(* IEC 61131-3 sources: Mizera_Tube/Plc (part 8) *)

END_VAR

VAR_OUTPUT
yax_READY:    BOOL;       * FB pronto per START
yax_RUNNING:  BOOL;       * Esecuzione FB in corso
yax_ENDOK:    BOOL;       * Comando terminato correttamente
yax_ENDERR:   BOOL;       * Comando terminato non correttamente
yax_ERRCODE:  DWORD;      * codice errore ( maschera bit )
END_VAR

VAR
AXFB: AX_COMMAND;
END_VAR

* Chiamata FB standard gestione comandi slave

LD   xax_ENABLE                    ** abilita FB
ST   AXFB.xax_ENABLE

LD   xax_START                     ** start richiesta azione
ST   AXFB.xax_START

LD   xax_CLEAR                     ** conferma fine comando
ST   AXFB.xax_CLEAR

CAL  AXFB

* Comando uscite da FB standard

LD   AXFB.yax_READY
ST   yax_READY                     ** FB pronto per START

LD   AXFB.yax_RUNNING
ST   yax_RUNNING                   ** Esecuzione FB in corso

LD   AXFB.yax_ENDOK
ST   yax_ENDOK                     ** Comando terminato correttamente

LD   AXFB.yax_ENDERR
ST   yax_ENDERR                    ** Comando terminato non correttamente

LD   AXFB.yax_ERRCODE
ST   yax_ERRCODE                   ** codice errore ( maschera bit )

*** TRASFERIMENTO DEI REGISTRI FB ALLO SLAVE ***

LD   AXFB.yax_RUNSLV
JMPCN END_DATA

LD   29
ST   FB_CODE                       ** fb0 Codice Operativo comando

LD   xax_NODE                      ** Numero nodo richiesto (2-60) o maschera
ST   %fb1

LD   xax_MODE                      ** Tipo di comando
ST   %fb2

END_DATA:

END_FUNCTION_BLOCK

* ----------------------------------------------------*
* Blocco Funzionale abilita/disabilita operatore dinamico su un asse
* ----------------------------------------------------*

FUNCTION_BLOCK AX_COUP

VAR_INPUT
xax_ENABLE:   BOOL;       * abilita FB
xax_START:    BOOL;       * start richiesta azione
xax_CLEAR:    BOOL;       * conferma fine comando
xax_MODE:     DWORD;      * Funzione selezionata
xax_INSTANCE: DWORD;      * Numero istanza tabella dati
xax_MASTER0:  DWORD;      * Numero asse master 0
xax_MASTER1:  DWORD;      * Numero asse master 1
xax_MASTER2:  DWORD;      * Numero asse master 2
xax_MASTER3:  DWORD;      * Numero asse master 3
xax_MASTER4:  DWORD;      * Numero asse master 4
xax_MASTER5:  DWORD;      * Numero asse master 5

END_VAR

VAR_OUTPUT
yax_READY:    BOOL;       * FB pronto per START
yax_RUNNING:  BOOL;       * Esecuzione FB in corso
yax_ENDOK:    BOOL;       * Comando terminato correttamente
yax_ENDERR:   BOOL;       * Comando terminato non correttamente
yax_ERRCODE:  DWORD;      * codice errore ( maschera bit )
END_VAR

VAR
AXFB: AX_COMMAND;
END_VAR

* Chiamata FB standard gestione comandi slave

LD   xax_ENABLE                    ** abilita FB
ST   AXFB.xax_ENABLE

LD   xax_START                     ** start richiesta azione
ST   AXFB.xax_START

LD   xax_CLEAR                     ** conferma fine comando
ST   AXFB.xax_CLEAR

CAL  AXFB

* Comando uscite da FB standard

LD   AXFB.yax_READY
ST   yax_READY                     ** FB pronto per START

LD   AXFB.yax_RUNNING
ST   yax_RUNNING                   ** Esecuzione FB in corso

LD   AXFB.yax_ENDOK
ST   yax_ENDOK                     ** Comando terminato correttamente

LD   AXFB.yax_ENDERR
ST   yax_ENDERR                    ** Comando terminato non correttamente

LD   AXFB.yax_ERRCODE
ST   yax_ERRCODE                   ** codice errore ( maschera bit )

*** TRASFERIMENTO DEI REGISTRI FB ALLO SLAVE ***

LD   AXFB.yax_TRDATA
JMPCN END_DATA

LD   31
ST   FB_CODE                       ** fb0 Codice Operativo comando

LD   xax_MODE                      ** Funzione selezionata
ST   FB_QUOTA                      ** fb1 Quota target assoluta (0.001 mm)

LD   xax_INSTANCE                  ** Numero istanza tabella dati
ST   FB_VEL                        ** fb2 Velocita' posizionamento (mm/min)

LD   xax_MASTER0                   ** Numero asse master 0
ST   FB_VMAX                       ** fb3 Velocita' massima (mm/min)

LD   xax_MASTER1                   ** Numero asse master 1
ST   FB_ACCEL                      ** fb4 Accelerazione (msec o mm/s2)

LD   xax_MASTER2                   ** Numero asse master 2
ST   FB_DECEL                      ** fb5 Decelerazione (msec o mm/s2)

LD   xax_MASTER3                   ** Numero asse master 3
ST   FB_RAMPES                     ** fb6 Tempo Rampe S (msec o mm/s3)

LD   xax_MASTER4                   ** Numero asse master 4
ST   FB_TOLLP                      ** fb7 Tolleranza (0.001 mm)

LD   xax_MASTER5                   ** Numero asse master 5
ST   FB_GAINP                      ** fb8 Guadagno P (0.001 DAC/pulses o 0.001 sec-1)

END_DATA:

END_FUNCTION_BLOCK

*******************************************************************************
*   FB gestione FC minimo/massimo e FC di taratura
*******************************************************************************
FUNCTION_BLOCK AX_LS_REF

VAR_INPUT
x_TYPE_LS:      DWORD;      * (1=NC, 0=NO)
x_REF_mode:     DWORD;      * 0=use ref switch NO
                            * 1=use ref switch NC
                            * 2=use MAX limit switch
                            * 3=use MIN limit switch
x_MIN_LS:       BOOL;       * Min Limit switch
x_MAX_LS:       BOOL;       * Max Limit switch
x_REF_S:        BOOL;       * Reference switch
END_VAR

VAR_OUTPUT
y_MIN_LS:       BOOL;       * Min Limit switch
y_MAX_LS:       BOOL;       * Max Limit switch
y_REF_S:        BOOL;       * Reference switch
END_VAR

VAR
l_MIN_LS:       BOOL;       * Min Limit switch
l_MAX_LS:       BOOL;       * Max Limit switch
l_REF_S:        BOOL;       * Reference switch
END_VAR
*******************************************************************************

LD   x_MIN_LS                      ** Min Limit switch
ST   l_MIN_LS                      ** Min Limit switch

LD   x_MAX_LS                      ** Max Limit switch
ST   l_MAX_LS                      ** Max Limit switch

LD   x_REF_S                       ** Reference switch
ST   l_REF_S                       ** Reference switch

LD   x_TYPE_LS                     ** (1=NC, 0=NO)
EQ   1
JMPCN NoNClose

LD   l_MIN_LS                      ** Min Limit switch
XOR  1
ST   l_MIN_LS                      ** Min Limit switch

LD   l_MAX_LS                      ** Max Limit switch
XOR  1
ST   l_MAX_LS                      ** Max Limit switch

NoNClose:
LD   x_REF_mode                    ** 0=use ref switch NO
EQ   0
JMPC exit_0

LD   x_REF_mode                    ** 0=use ref switch NO
EQ   1
JMPCN check_v2

LD   x_REF_S                       ** Reference switch
XOR  1
ST   l_REF_S                       ** Reference switch
JMP  exit_0

*****************************
*   FC +
*****************************
check_v2:
LD   x_REF_mode                    ** 0=use ref switch NO
EQ   2
JMPCN check_v3

LD   %ui16.1                        ** Selezione Modo REF da Plc
JMPCN check_v3

LD   ALWAYS_ZERO                   ** PLCFLAGS.0  Flag sempre stato off
ST   l_MAX_LS                      ** Max Limit switch

LD   x_TYPE_LS                     ** (1=NC, 0=NO)
EQ   1                              ** nc condition
JMPCN no_switch

LDN  x_MAX_LS                      ** Max Limit switch
ST   l_REF_S                       ** Reference switch

JMP  exit_0
no_switch:

LD   x_MAX_LS                      ** Max Limit switch
ST   l_REF_S                       ** Reference switch

JMP  exit_0

*****************************
*   FC -
*****************************
check_v3:
LD   x_REF_mode                    ** 0=use ref switch NO
EQ   3
JMPCN check_v4

LD   %ui16.1                        ** Selezione Modo REF da Plc
JMPCN check_v4

LD   ALWAYS_ZERO                   ** PLCFLAGS.0  Flag sempre stato off
ST   l_MIN_LS                      ** Min Limit switch

LD   x_TYPE_LS                     ** (1=NC, 0=NO)
EQ   1                              ** nc condition
JMPCN no_switch1

LDN  x_MIN_LS                      ** Min Limit switch
ST   l_REF_S                       ** Reference switch

JMP  exit_0
no_switch1:

LD   x_MIN_LS                      ** Min Limit switch
ST   l_REF_S                       ** Reference switch

JMP  exit_0

check_v4:
exit_0:
LD   l_MIN_LS                      ** Min Limit switch
ST   y_MIN_LS                      ** Min Limit switch

LD   l_MAX_LS                      ** Max Limit switch
ST   y_MAX_LS                      ** Max Limit switch

LD   l_REF_S                       ** Reference switch
ST   y_REF_S                       ** Reference switch
JMP  exit_com

exit_com:

END_FUNCTION_BLOCK

(* ---- AxTrack.plc ---- *)
*//============================================================================
*// AXIS TRACKING FROM PLC
*//============================================================================
* Only Used during program running
*
* CAL SEGUI_AXIS0(xAxNum:=,xMove:=,xTarget:=,xSpeed:=)
*
* LD  SEGUI_AXIS0.yFromPlc
* ST  GESTAX*.xFromPlc
*//============================================================================

#funcdec "assi.plc"
#funcdec "cnc.plc"
#include "iol.inc"

VAR
#include "assi.inc"
#include "cnc.inc"
#include "mem.inc"
END_VAR

FUNCTION_BLOCK  AX_VAR_TRACK

*//============================================================================
* To keep axis following target
*//============================================================================

VAR_INPUT
xAxNum:            DWORD;         * Axis ID
xMove:             BOOL;          * Move CMD
xTarget:           DWORD;         * Destination
xSpeed:            DWORD;         * Moving Speed
END_VAR

VAR_OUTPUT
yFromPlc:          BOOL;
END_VAR

VAR
TP_PRGOFF:         TP;
TOF_RESET:         TOF;
Appoggio:          BOOL;
POS_AX:            AX_SINGVAR;
END_VAR

PATH %ax[xAxNum]

*//============================================================================

LD   xMove
AND  MACC_TARATA
ANDN EMER_GEN
ANDN MACC_ALARM
AND  %cn0.rc8.0
ANDN %cn0.rc8.1
ST   POS_AX.xax_ENABLE
ST   yFromPlc

LDN  %cn0.rc8.0
ST   Appoggio
CAL  TP_PRGOFF(IN=Appoggio, PT=10)
CAL  TOF_RESET(IN=Pul_Reset, PT=10)

LDN  POS_AX.xax_ENABLE
OR   TP_PRGOFF.Q
OR   TOF_RESET.Q
ST   POS_AX.xax_CLEAR

LD   POS_AX.xax_ENABLE
AND  POS_AX.yax_READY
ANDN POS_AX.yax_ENDERR
ST   POS_AX.xax_START

LD   xTarget
ST   POS_AX.xax_QUOTA

LD   xSpeed
ST   POS_AX.xax_VEL

CAL  POS_AX

*//============================================================================

END_FUNCTION_BLOCK

(* ---- Canfb.plc ---- *)
* Blocchi gestione periferiche CANopen da PLC

VAR_IN_OUT
AS_DATA0 AT %CanFb48; * CanFb48 buffer I/O Canopen
AS_DATA1 AT %CanFb49; * CanFb49 buffer I/O Canopen
AS_DATA2 AT %CanFb50; * CanFb50 buffer I/O Canopen
AS_DATA3 AT %CanFb51; * CanFb51 buffer I/O Canopen
AS_DATA4 AT %CanFb52; * CanFb52 buffer I/O Canopen
AS_DATA5 AT %CanFb53; * CanFb53 buffer I/O Canopen
AS_DATA6 AT %CanFb54; * CanFb54 buffer I/O Canopen
AS_DATA7 AT %CanFb55; * CanFb55 buffer I/O Canopen
DI_DATA0 AT %CanFb56; * CanFb56 Dato 0 input
DI_DATA1 AT %CanFb57; * CanFb57 Dato 1 input
DI_COBID AT %CanFb58; * CanFb58 Identificatore oggetto CanOpen
CONTROLREG AT %CanFb59; * CanFb59 registro comando (bit 0-7=codice comando)
CMD_RESET AT %CanFb59.30; * CanFb59.30 Reset nodo
CMD_ENAB AT %CanFb59.31; * CanFb59.31 Enable esecuzione comando
STATUSREG AT %CanFb60; * CanFb60 registro stato
DO_CONFIRM AT %CanFb60.31; * CanFb60.31 conferma comando eseguito
DO_ERROR AT %CanFb61; * CanFb61 codice errore comando
DO_DATA0 AT %CanFb62; * CanFb62 Dato 0 output
DO_DATA1 AT %CanFb63; * CanFb63 Dato 1 output
END_VAR

* -------------------------------------------------------*
* Blocco Funzionale generico invio comando a nodo CANopen
* -------------------------------------------------------*

FUNCTION_BLOCK COP_COMMAND

VAR_INPUT
CM_ENAB: BOOL; * Richiesta esecuzione comando
CM_RESET: BOOL; * Richiesta di reset del nodo
CM_CODE: DWORD; * Codice del comando
CI_COBID: DWORD; * Identificatore oggetto CanOpen
CI_DATA0: DWORD; * Dato 0 in input
CI_DATA1: DWORD; * Dato 1 in input
END_VAR

VAR_OUTPUT
CS_CONFIRM: BOOL; * Conferma comando eseguito
CO_ERROR: WORD; * Codice di errore
CO_ERRORINFO: DWORD; * Informazioni aggiuntive su errore
CO_DATA0: DWORD; * Dato 0 in output
CO_DATA1: DWORD; * Dato 1 in output
CO_DATA2: DWORD; * Dato 2 in output
CO_DATA3: DWORD; * Dato 3 in output
CO_DATA4: DWORD; * Dato 4 in output
CO_DATA5: DWORD; * Dato 5 in output
CO_DATA6: DWORD; * Dato 6 in output
CO_DATA7: DWORD; * Dato 7 in output
CO_DATA8: DWORD; * Dato 8 in output
END_VAR

VAR
StPrecEnab: BOOL; * Stato precedente ingresso ENAB
StPrecReset: BOOL; * Stato precedente ingresso RESET
StPrecConfirm: BOOL; * Stato precedente segnale CONFIRM
RTEnab: BOOL; * Fronte salita ingresso ENAB
MemCmdInProg: BOOL; * Mem. comando in corso
MemErrBusy: BOOL; * Mem. errore area comandi occupata
CmdFinished: BOOL; * Conferma comando terminato
END_VAR

* Sul fronte di salita del comando, copia tutti i dati in andata

LD   CM_ENAB                       ** Richiesta esecuzione comando
ANDN StPrecEnab                    ** Stato precedente ingresso ENAB
ST   RTEnab                        ** Fronte salita ingresso ENAB

LD   RTEnab                        ** Fronte salita ingresso ENAB
ANDN CMD_ENAB                      ** CanFb59.31 Enable esecuzione comando
ANDN DO_CONFIRM                    ** CanFb60.31 conferma comando eseguito
S    MemCmdInProg                  ** Mem. comando in corso

LDN  CM_ENAB                       ** Richiesta esecuzione comando
ANDN CMD_ENAB                      ** CanFb59.31 Enable esecuzione comando
ANDN DO_CONFIRM                    ** CanFb60.31 conferma comando eseguito
OR   CM_RESET                      ** Richiesta di reset del nodo
R    MemCmdInProg                  ** Mem. comando in corso

LD   RTEnab                        ** Fronte salita ingresso ENAB
ANDN MemCmdInProg                  ** Mem. comando in corso
S    MemErrBusy                    ** Mem. errore area comandi occupata

LDN  CM_ENAB                       ** Richiesta esecuzione comando
R    MemErrBusy                    ** Mem. errore area comandi occupata

LD   RTEnab                        ** Fronte salita ingresso ENAB
AND  MemCmdInProg                  ** Mem. comando in corso
JMPCN END_COMMAND

LD   CONTROLREG                    ** CanFb59 registro comando (bit 0-7=codice comando)
AND  16#FFFFFF00
OR   CM_CODE                       ** Codice del comando
ST   CONTROLREG                    ** CanFb59 registro comando (bit 0-7=codice comando)

LD   CI_COBID                      ** Identificatore oggetto CanOpen
ST   DI_COBID                      ** CanFb58 Identificatore oggetto CanOpen

LD   CM_CODE                       ** Codice del comando
EQ   4            * PDO SEND
JMPC PDO_SEND_CMD

LD   CI_DATA0                      ** Dato 0 in input
ST   DI_DATA0                      ** CanFb56 Dato 0 input

LD   CI_DATA1                      ** Dato 1 in input
ST   DI_DATA1                      ** CanFb57 Dato 1 input

JMP  END_COMMAND

PDO_SEND_CMD:
LD   DI_COBID                      ** CanFb58 Identificatore oggetto CanOpen
AND  16#FFFF00FF  * Mask offset
OR   16#3000      * Offset AS_DATA0 (48)
ST   DI_COBID                      ** CanFb58 Identificatore oggetto CanOpen

LD   CI_DATA0                      ** Dato 0 in input
ST   AS_DATA0                      ** CanFb48 buffer I/O Canopen

LD   CI_DATA1                      ** Dato 1 in input
ST   AS_DATA1                      ** CanFb49 buffer I/O Canopen

END_COMMAND:

LD   CM_ENAB                       ** Richiesta esecuzione comando
ST   StPrecEnab                    ** Stato precedente ingresso ENAB

* Scrive i bit di ENAB e RESET

LD   MemCmdInProg                  ** Mem. comando in corso
JMPCN END_CMD_ENAB

LD   CM_ENAB                       ** Richiesta esecuzione comando
ST   CMD_ENAB                      ** CanFb59.31 Enable esecuzione comando

END_CMD_ENAB:

LD   CM_RESET                      ** Richiesta di reset del nodo
OR   StPrecReset                   ** Stato precedente ingresso RESET
JMPCN END_RESET

LD   CM_RESET                      ** Richiesta di reset del nodo
ST   CMD_RESET                     ** CanFb59.30 Reset nodo

LD   %PLCFLAGS.0
ST   CMD_ENAB                      ** CanFb59.31 Enable esecuzione comando

END_RESET:

LD   CM_RESET                      ** Richiesta di reset del nodo
ST   StPrecReset                   ** Stato precedente ingresso RESET

* Sul fronte di salita della conferma fine comando, legge tutti i dati di ritorno

LD   DO_CONFIRM                    ** CanFb60.31 conferma comando eseguito
AND  MemCmdInProg                  ** Mem. comando in corso
ST   CmdFinished                   ** Conferma comando terminato

LD   DO_CONFIRM                    ** CanFb60.31 conferma comando eseguito
ANDN StPrecConfirm                 ** Stato precedente segnale CONFIRM
AND  CmdFinished                   ** Conferma comando terminato
JMPCN END_DATA

LD   DO_ERROR                      ** CanFb61 codice errore comando
ST   CO_ERROR                      ** Codice di errore

LD   DO_ERROR                      ** CanFb61 codice errore comando
NE   0
JMPC TAKE_ERRINFO

LD   0
ST   CO_ERRORINFO                  ** Informazioni aggiuntive su errore

LD   CM_CODE                       ** Codice del comando
EQ   5            * PDO READ
OR   (
LD   CM_CODE                       ** Codice del comando
EQ   9            * SDO READSTR
)
OR   (
LD   CM_CODE                       ** Codice del comando
EQ   10           * HISTORY ALARM
)
JMPC PDO_READ_CMD

LD   DO_DATA0                      ** CanFb62 Dato 0 output
ST   CO_DATA0                      ** Dato 0 in output

LD   DO_DATA1                      ** CanFb63 Dato 1 output
ST   CO_DATA1                      ** Dato 1 in output

JMP  END_DATA

PDO_READ_CMD:

LD   DO_DATA0                      ** CanFb62 Dato 0 output
ST   CO_DATA0                      ** Dato 0 in output

LD   AS_DATA0                      ** CanFb48 buffer I/O Canopen
ST   CO_DATA1                      ** Dato 1 in output

LD   AS_DATA1                      ** CanFb49 buffer I/O Canopen
ST   CO_DATA2                      ** Dato 2 in output

LD   CM_CODE                       ** Codice del comando
EQ   5            * PDO READ
JMPC END_DATA

LD   AS_DATA2                      ** CanFb50 buffer I/O Canopen
ST   CO_DATA3                      ** Dato 3 in output

LD   AS_DATA3                      ** CanFb51 buffer I/O Canopen
ST   CO_DATA4                      ** Dato 4 in output

LD   AS_DATA4                      ** CanFb52 buffer I/O Canopen
ST   CO_DATA5                      ** Dato 5 in output

LD   AS_DATA5                      ** CanFb53 buffer I/O Canopen
ST   CO_DATA6                      ** Dato 6 in output

LD   AS_DATA6                      ** CanFb54 buffer I/O Canopen
ST   CO_DATA7                      ** Dato 7 in output

LD   AS_DATA7                      ** CanFb55 buffer I/O Canopen
ST   CO_DATA8                      ** Dato 8 in output

JMP  END_DATA

TAKE_ERRINFO:

LD   DO_DATA0                      ** CanFb62 Dato 0 output
ST   CO_ERRORINFO                  ** Informazioni aggiuntive su errore

LD   0
ST   CO_DATA0                      ** Dato 0 in output
ST   CO_DATA1                      ** Dato 1 in output

END_DATA:

LD   MemErrBusy                    ** Mem. errore area comandi occupata
JMPCN END_TR_ERR

LD   16#25        * Errore TRANSFER_BUSY
ST   CO_ERROR                      ** Codice di errore

END_TR_ERR:

* Scrive in output la conferma

LD   DO_CONFIRM                    ** CanFb60.31 conferma comando eseguito
ST   StPrecConfirm                 ** Stato precedente segnale CONFIRM

LD   CmdFinished                   ** Conferma comando terminato
OR   MemErrBusy                    ** Mem. errore area comandi occupata
ST   CS_CONFIRM                    ** Conferma comando eseguito

END_FUNCTION_BLOCK

* -------------------------------------------------------*
* Comando di cambio di stato a nodo CANopen
* -------------------------------------------------------*

FUNCTION_BLOCK COP_NMT

VAR_INPUT
CM_ENAB: BOOL; * Richiesta esecuzione comando
CM_RESET: BOOL; * Richiesta di reset del nodo
CI_STATE: DWORD; * Stato richiesto
END_VAR

VAR_OUTPUT
CS_CONFIRM: BOOL; * Conferma comando eseguito
CO_ERROR: WORD; * Codice di errore
END_VAR

VAR
COPFB: COP_COMMAND;
END_VAR

LD   CM_ENAB                       ** Richiesta esecuzione comando
ST   COPFB.CM_ENAB

LD   CM_RESET                      ** Richiesta di reset del nodo
ST   COPFB.CM_RESET

LD   1
ST   COPFB.CM_CODE

LD   CI_STATE                      ** Stato richiesto
ST   COPFB.CI_DATA0

CAL  COPFB

LD   COPFB.CS_CONFIRM
ST   CS_CONFIRM                    ** Conferma comando eseguito

LD   COPFB.CO_ERROR
ST   CO_ERROR                      ** Codice di errore

END_FUNCTION_BLOCK

* -------------------------------------------------------*
* Comando di lettura SDO a nodo CANopen
* -------------------------------------------------------*

FUNCTION_BLOCK COP_SDO_READ

VAR_INPUT
CM_ENAB: BOOL; * Richiesta esecuzione comando
CM_RESET: BOOL; * Richiesta di reset del nodo
CI_INDEX: DWORD; * Numero index dato da leggere
CI_SUBINDEX: DWORD; * Numero subindex dato da leggere
END_VAR

VAR_OUTPUT
CS_CONFIRM: BOOL; * Conferma comando eseguito
CO_ERROR: WORD; * Codice di errore
CO_ERRORINFO: DWORD; * Informazioni aggiuntive su errore
CO_DATALENGTH: DWORD; * Lunghezza dato letto in byte
CO_DATA0: DWORD; * Valore del dato letto
END_VAR

VAR
COPFB: COP_COMMAND;
END_VAR

LD   CM_ENAB                       ** Richiesta esecuzione comando
ST   COPFB.CM_ENAB

LD   CM_RESET                      ** Richiesta di reset del nodo
ST   COPFB.CM_RESET

LD   2
ST   COPFB.CM_CODE

LD   CI_INDEX                      ** Numero index dato da leggere
SHL  16
OR   (
LD   CI_SUBINDEX                   ** Numero subindex dato da leggere
SHL  8
)
ST   COPFB.CI_COBID

CAL  COPFB

LD   COPFB.CS_CONFIRM
ST   CS_CONFIRM                    ** Conferma comando eseguito

LD   COPFB.CO_ERROR
ST   CO_ERROR                      ** Codice di errore

LD   COPFB.CO_ERRORINFO
ST   CO_ERRORINFO                  ** Informazioni aggiuntive su errore

LD   COPFB.CO_DATA0
ST   CO_DATALENGTH                 ** Lunghezza dato letto in byte

LD   COPFB.CO_DATA1
ST   CO_DATA0                      ** Valore del dato letto

END_FUNCTION_BLOCK

* -------------------------------------------------------*
* Comando di scrittura SDO a nodo CANopen
* -------------------------------------------------------*

FUNCTION_BLOCK COP_SDO_WRITE

VAR_INPUT
CM_ENAB: BOOL; * Richiesta esecuzione comando
CM_RESET: BOOL; * Richiesta di reset del nodo
CI_INDEX: DWORD; * Numero index dato da scrivere
CI_SUBINDEX: DWORD; * Numero subindex dato da scrivere
CI_DATALENGTH: DWORD; * Lunghezza dato da scrivere in byte
CI_DATA0: DWORD; * Valore da scrivere
END_VAR

VAR_OUTPUT
CS_CONFIRM: BOOL; * Conferma comando eseguito
CO_ERROR: WORD; * Codice di errore
CO_ERRORINFO: DWORD; * Informazioni aggiuntive su errore
END_VAR

VAR
COPFB: COP_COMMAND;
END_VAR

LD   CM_ENAB                       ** Richiesta esecuzione comando
ST   COPFB.CM_ENAB

LD   CM_RESET                      ** Richiesta di reset del nodo
ST   COPFB.CM_RESET

LD   3
ST   COPFB.CM_CODE

LD   CI_INDEX                      ** Numero index dato da scrivere
SHL  16
OR   (
LD   CI_SUBINDEX                   ** Numero subindex dato da scrivere
SHL  8
)
OR   CI_DATALENGTH                 ** Lunghezza dato da scrivere in byte
ST   COPFB.CI_COBID

LD   CI_DATA0                      ** Valore da scrivere
ST   COPFB.CI_DATA0

CAL  COPFB

LD   COPFB.CS_CONFIRM
ST   CS_CONFIRM                    ** Conferma comando eseguito

LD   COPFB.CO_ERROR
ST   CO_ERROR                      ** Codice di errore

LD   COPFB.CO_ERRORINFO
ST   CO_ERRORINFO                  ** Informazioni aggiuntive su errore

END_FUNCTION_BLOCK

* -------------------------------------------------------*
* Comando di invio PDO a nodo CANopen
* -------------------------------------------------------*

FUNCTION_BLOCK COP_PDO_SEND

VAR_INPUT
CM_ENAB: BOOL; * Richiesta esecuzione comando
CM_RESET: BOOL; * Richiesta di reset del nodo
CI_COBID: DWORD; * Identificatore oggetto CanOpen
CI_DATALENGTH: DWORD; * Lunghezza dato da scrivere in byte
CI_DATA0: DWORD; * Valore da inviare (BYTE 0-3)
CI_DATA1: DWORD; * Valore da inviare (BYTE 4-7)
END_VAR

VAR_OUTPUT
CS_CONFIRM: BOOL; * Conferma comando eseguito
CO_ERROR: WORD; * Codice di errore
END_VAR

VAR
COPFB: COP_COMMAND;
END_VAR

LD   CM_ENAB                       ** Richiesta esecuzione comando
ST   COPFB.CM_ENAB

LD   CM_RESET                      ** Richiesta di reset del nodo
ST   COPFB.CM_RESET

LD   4
ST   COPFB.CM_CODE

LD   CI_COBID                      ** Identificatore oggetto CanOpen
SHL  16
OR   CI_DATALENGTH                 ** Lunghezza dato da scrivere in byte
ST   COPFB.CI_COBID

LD   CI_DATA0                      ** Valore da inviare (BYTE 0-3)
ST   COPFB.CI_DATA0

LD   CI_DATA1                      ** Valore da inviare (BYTE 4-7)
ST   COPFB.CI_DATA1

CAL  COPFB

LD   COPFB.CS_CONFIRM
ST   CS_CONFIRM                    ** Conferma comando eseguito

LD   COPFB.CO_ERROR
ST   CO_ERROR                      ** Codice di errore

END_FUNCTION_BLOCK

* -------------------------------------------------------*
* Comando di lettura PDO da nodo CANopen
* -------------------------------------------------------*

FUNCTION_BLOCK COP_PDO_READ

VAR_INPUT
CM_ENAB: BOOL; * Richiesta esecuzione comando
CM_RESET: BOOL; * Richiesta di reset del nodo
CI_COBID: DWORD; * Identificatore oggetto CanOpen
END_VAR

VAR_OUTPUT
CS_CONFIRM: BOOL; * Conferma comando eseguito
CO_ERROR: WORD; * Codice di errore
CO_DATALENGTH: DWORD; * Lunghezza PDO letto in byte
CO_DATA0: DWORD; * Valore del dato letto (BYTE 0-3)
CO_DATA1: DWORD; * Valore del dato letto (BYTE 4-7)
END_VAR

VAR
COPFB: COP_COMMAND;
END_VAR

LD   CM_ENAB                       ** Richiesta esecuzione comando
ST   COPFB.CM_ENAB

LD   CM_RESET                      ** Richiesta di reset del nodo
ST   COPFB.CM_RESET

LD   5
ST   COPFB.CM_CODE

LD   CI_COBID                      ** Identificatore oggetto CanOpen
SHL  16
ST   COPFB.CI_COBID

CAL  COPFB

LD   COPFB.CS_CONFIRM
ST   CS_CONFIRM                    ** Conferma comando eseguito

LD   COPFB.CO_ERROR
ST   CO_ERROR                      ** Codice di errore

LD   COPFB.CO_DATA0
ST   CO_DATALENGTH                 ** Lunghezza PDO letto in byte

LD   COPFB.CO_DATA1
ST   CO_DATA0                      ** Valore del dato letto (BYTE 0-3)

LD   COPFB.CO_DATA2
ST   CO_DATA1                      ** Valore del dato letto (BYTE 4-7)

END_FUNCTION_BLOCK

* -------------------------------------------------------*
* Comando di registrazione PDO
* -------------------------------------------------------*

FUNCTION_BLOCK COP_PDO_REGISTER

VAR_INPUT
CM_ENAB: BOOL; * Richiesta esecuzione comando
CM_RESET: BOOL; * Richiesta di reset del nodo
CI_COBID: DWORD; * Identificatore oggetto CanOpen
CI_DATALENGTH: DWORD; * Lunghezza in BYTE e tipo dato (FFFF = cancella registr.)
                      * lungh + 0: legge con COP_PDO_READ
                      * lungh + 256: legge da CanFb0-CanFb47
                      * lungh + 512: legge da IW0-IW2047
CI_DATAOFFSET: DWORD; * Offset rinfresco (CanFb[0-47] / IO[0-2047])
END_VAR

VAR_OUTPUT
CS_CONFIRM: BOOL; * Conferma comando eseguito
CO_ERROR: WORD; * Codice di errore
END_VAR

VAR
COPFB: COP_COMMAND;
END_VAR

LD   CM_ENAB                       ** Richiesta esecuzione comando
ST   COPFB.CM_ENAB

LD   CM_RESET                      ** Richiesta di reset del nodo
ST   COPFB.CM_RESET

LD   6
ST   COPFB.CM_CODE

LD   CI_COBID                      ** Identificatore oggetto CanOpen
SHL  16
OR   CI_DATALENGTH                 ** Lunghezza in BYTE e tipo dato (FFFF = cancella registr.)
ST   COPFB.CI_COBID

LD   CI_DATAOFFSET                 ** Offset rinfresco (CanFb[0-47] / IO[0-2047])
ST   COPFB.CI_DATA0

CAL  COPFB

LD   COPFB.CS_CONFIRM
ST   CS_CONFIRM                    ** Conferma comando eseguito

LD   COPFB.CO_ERROR
ST   CO_ERROR                      ** Codice di errore

END_FUNCTION_BLOCK

* -------------------------------------------------------*
* Comando di impostazione sincronizzazione ciclica
* -------------------------------------------------------*

FUNCTION_BLOCK COP_CYCLIC_SYNC

VAR_INPUT
CM_ENAB: BOOL; * Richiesta esecuzione comando
CM_RESET: BOOL; * Richiesta di reset del nodo
CI_SYNC_TIME: DWORD; * Tempo ciclo (0=Disab, 1=Singolo, 10-250=Ciclico in ms)
END_VAR

VAR_OUTPUT
CS_CONFIRM: BOOL; * Conferma comando eseguito
CO_ERROR: WORD; * Codice di errore
END_VAR

VAR
COPFB: COP_COMMAND;
END_VAR

LD   CM_ENAB                       ** Richiesta esecuzione comando
ST   COPFB.CM_ENAB

LD   CM_RESET                      ** Richiesta di reset del nodo
ST   COPFB.CM_RESET

LD   7
ST   COPFB.CM_CODE

LD   CI_SYNC_TIME                  ** Tempo ciclo (0=Disab, 1=Singolo, 10-250=Ciclico in ms)
ST   COPFB.CI_DATA0

CAL  COPFB

LD   COPFB.CS_CONFIRM
ST   CS_CONFIRM                    ** Conferma comando eseguito

LD   COPFB.CO_ERROR
ST   CO_ERROR                      ** Codice di errore

END_FUNCTION_BLOCK

* -------------------------------------------------------*
* Comando di remote request oggetto CANopen
* -------------------------------------------------------*

FUNCTION_BLOCK COP_REM_REQUEST

VAR_INPUT
CM_ENAB: BOOL; * Richiesta esecuzione comando
CM_RESET: BOOL; * Richiesta di reset del nodo
CI_COBID: DWORD; * Identificatore oggetto CanOpen
END_VAR

VAR_OUTPUT
CS_CONFIRM: BOOL; * Conferma comando eseguito
CO_ERROR: WORD; * Codice di errore
END_VAR

VAR
COPFB: COP_COMMAND;
END_VAR

LD   CM_ENAB                       ** Richiesta esecuzione comando
ST   COPFB.CM_ENAB

LD   CM_RESET                      ** Richiesta di reset del nodo
ST   COPFB.CM_RESET

LD   8
ST   COPFB.CM_CODE

LD   CI_COBID                      ** Identificatore oggetto CanOpen
ST   COPFB.CI_COBID

CAL  COPFB

LD   COPFB.CS_CONFIRM
ST   CS_CONFIRM                    ** Conferma comando eseguito

LD   COPFB.CO_ERROR
ST   CO_ERROR                      ** Codice di errore

END_FUNCTION_BLOCK

* -------------------------------------------------------*
* Comando di lettura SDO su stringa da nodo CANopen
* -------------------------------------------------------*

FUNCTION_BLOCK COP_SDO_READSTRING

VAR_INPUT
CM_ENAB: BOOL; * Richiesta esecuzione comando
CM_RESET: BOOL; * Richiesta di reset del nodo
CI_INDEX: DWORD; * Numero index dato da leggere
CI_SUBINDEX: DWORD; * Numero subindex dato da leggere
END_VAR

VAR_OUTPUT
CS_CONFIRM: BOOL; * Conferma comando eseguito
CO_ERROR: WORD; * Codice di errore
CO_ERRORINFO: DWORD; * Informazioni aggiuntive su errore
CO_DATALENGTH: DWORD; * Lunghezza stringa letta in byte
CO_DATA0: DWORD; * Stringa letta (BYTE 0-3)
CO_DATA1: DWORD; * Stringa letta (BYTE 4-7)
CO_DATA2: DWORD; * Stringa letta (BYTE 8-11)
CO_DATA3: DWORD; * Stringa letta (BYTE 12-15)
CO_DATA4: DWORD; * Stringa letta (BYTE 16-19)
CO_DATA5: DWORD; * Stringa letta (BYTE 20-23)
CO_DATA6: DWORD; * Stringa letta (BYTE 24-27)
CO_DATA7: DWORD; * Stringa letta (BYTE 28-31)
END_VAR

VAR
COPFB: COP_COMMAND;
END_VAR

LD   CM_ENAB                       ** Richiesta esecuzione comando
ST   COPFB.CM_ENAB

LD   CM_RESET                      ** Richiesta di reset del nodo
ST   COPFB.CM_RESET

LD   9
ST   COPFB.CM_CODE

LD   CI_INDEX                      ** Numero index dato da leggere
SHL  16
OR   (
LD   CI_SUBINDEX                   ** Numero subindex dato da leggere
SHL  8
)
ST   COPFB.CI_COBID

CAL  COPFB

LD   COPFB.CS_CONFIRM
ST   CS_CONFIRM                    ** Conferma comando eseguito

LD   COPFB.CO_ERROR
ST   CO_ERROR                      ** Codice di errore

LD   COPFB.CO_ERRORINFO
ST   CO_ERRORINFO                  ** Informazioni aggiuntive su errore

LD   COPFB.CO_DATA0
ST   CO_DATALENGTH                 ** Lunghezza stringa letta in byte

LD   COPFB.CO_DATA1
ST   CO_DATA0                      ** Stringa letta (BYTE 0-3)

LD   COPFB.CO_DATA2
ST   CO_DATA1                      ** Stringa letta (BYTE 4-7)

LD   COPFB.CO_DATA3
ST   CO_DATA2                      ** Stringa letta (BYTE 8-11)

LD   COPFB.CO_DATA4
ST   CO_DATA3                      ** Stringa letta (BYTE 12-15)

LD   COPFB.CO_DATA5
ST   CO_DATA4                      ** Stringa letta (BYTE 16-19)

LD   COPFB.CO_DATA6
ST   CO_DATA5                      ** Stringa letta (BYTE 20-23)

LD   COPFB.CO_DATA7
ST   CO_DATA6                      ** Stringa letta (BYTE 24-27)

LD   COPFB.CO_DATA8
ST   CO_DATA7                      ** Stringa letta (BYTE 28-31)

END_FUNCTION_BLOCK

* -------------------------------------------------------*
* Comando Read/Reset History alarm da nodo CANopen
* -------------------------------------------------------*

FUNCTION_BLOCK COP_ALARMS_HIST

VAR_INPUT
CM_ENAB:  BOOL; * Richiesta esecuzione comando
CM_RESET: BOOL; * Richiesta di reset del nodo
CI_MODE:  BOOL; * 0=Read  1=Read & Reset
END_VAR

VAR_OUTPUT
CS_CONFIRM: BOOL; * Conferma comando eseguito
CO_ERROR:   WORD; * Codice di errore
CO_ERRORINFO: DWORD;  * Informazioni aggiuntive su errore
CO_ALARMS:    DWORD;  * Numero di allarmi presenti
CO_ALRM1: DWORD; * Ultimo allarme "n"
CO_ALRM2: DWORD; * Allarme "n-1"
CO_ALRM3: DWORD; * Allarme "n-2"
CO_ALRM4: DWORD; * Allarme "n-3"
CO_ALRM5: DWORD; * Allarme "n-4"
CO_ALRM6: DWORD; * Allarme "n-5"
CO_ALRM7: DWORD; * Allarme "n-6"
CO_ALRM8: DWORD; * Allarme "n-7"
END_VAR

VAR
COPFB: COP_COMMAND;
END_VAR

LD   CM_ENAB                       ** Richiesta esecuzione comando
ST   COPFB.CM_ENAB

LD   CM_RESET                      ** Richiesta di reset del nodo
ST   COPFB.CM_RESET

LD   10
ST   COPFB.CM_CODE

LD   CI_MODE                       ** 0=Read  1=Read & Reset
ST   COPFB.CI_DATA0.0   ** CanFb56 Dato 0 input

CAL  COPFB

LD   COPFB.CS_CONFIRM
ST   CS_CONFIRM                    ** Conferma comando eseguito

LD   COPFB.CO_ERROR
ST   CO_ERROR                      ** Codice di errore

LD   COPFB.CO_ERRORINFO
ST   CO_ERRORINFO                  ** Informazioni aggiuntive su errore

LD   DO_DATA0                      ** CanFb62 Dato 0 output
ST   CO_ALARMS                     ** Numero di allarmi presenti

LD   COPFB.CO_DATA1
ST   CO_ALRM1                      ** Ultimo allarme "n"

LD   COPFB.CO_DATA2
ST   CO_ALRM2                      ** Allarme "n-1"

LD   COPFB.CO_DATA3
ST   CO_ALRM3                      ** Allarme "n-2"

LD   COPFB.CO_DATA4
ST   CO_ALRM4                      ** Allarme "n-3"

LD   COPFB.CO_DATA5
ST   CO_ALRM5                      ** Allarme "n-4"

LD   COPFB.CO_DATA6
ST   CO_ALRM6                      ** Allarme "n-5"

LD   COPFB.CO_DATA7
ST   CO_ALRM7                      ** Allarme "n-6"

LD   COPFB.CO_DATA8
ST   CO_ALRM8                      ** Allarme "n-7"

END_FUNCTION_BLOCK

* -------------------------------------------------------*
* Comando di lettura VACON ReadAnyParam
* -------------------------------------------------------*

FUNCTION_BLOCK VAC_PAR_READ

VAR_INPUT
CM_ENAB: BOOL; * Richiesta esecuzione comando
CM_RESET: BOOL; * Richiesta di reset del nodo
CI_INDEX: DWORD; * Numero parametro da leggere
END_VAR

VAR_OUTPUT
CS_CONFIRM: BOOL; * Conferma comando eseguito
CO_ERROR: WORD; * Codice di errore
CO_ERRORINFO: DWORD; * Informazioni aggiuntive su errore
CO_DATALENGTH: DWORD; * Lunghezza dato letto in byte
CO_DATA0: DWORD; * Valore del dato letto
END_VAR

VAR
COPFB: COP_COMMAND;
END_VAR

LD   CM_ENAB                       ** Richiesta esecuzione comando
ST   COPFB.CM_ENAB

LD   CM_RESET                      ** Richiesta di reset del nodo
ST   COPFB.CM_RESET

LD   255
ST   COPFB.CM_CODE

LD   CI_INDEX                      ** Numero parametro da leggere
ST   COPFB.CI_COBID

CAL  COPFB

LD   COPFB.CS_CONFIRM
ST   CS_CONFIRM                    ** Conferma comando eseguito

LD   COPFB.CO_ERROR
ST   CO_ERROR                      ** Codice di errore

LD   COPFB.CO_ERRORINFO
ST   CO_ERRORINFO                  ** Informazioni aggiuntive su errore

LD   COPFB.CO_DATA0
ST   CO_DATALENGTH                 ** Lunghezza dato letto in byte

LD   COPFB.CO_DATA1
ST   CO_DATA0                      ** Valore del dato letto

END_FUNCTION_BLOCK

* -------------------------------------------------------*
* Comando di scrittura VACON WriteAnyParam
* -------------------------------------------------------*

FUNCTION_BLOCK VAC_PAR_WRITE

VAR_INPUT
CM_ENAB: BOOL; * Richiesta esecuzione comando
CM_RESET: BOOL; * Richiesta di reset del nodo
CI_INDEX: DWORD; * Numero parametro dato da scrivere
CI_DATA0: DWORD; * Valore da scrivere
END_VAR

VAR_OUTPUT
CS_CONFIRM: BOOL; * Conferma comando eseguito
CO_ERROR: WORD; * Codice di errore
CO_ERRORINFO: DWORD; * Informazioni aggiuntive su errore
END_VAR

VAR
COPFB: COP_COMMAND;
END_VAR

LD   CM_ENAB                       ** Richiesta esecuzione comando
ST   COPFB.CM_ENAB

LD   CM_RESET                      ** Richiesta di reset del nodo
ST   COPFB.CM_RESET

LD   254
ST   COPFB.CM_CODE

LD   CI_INDEX                      ** Numero parametro dato da scrivere
ST   COPFB.CI_COBID

LD   CI_DATA0                      ** Valore da scrivere
ST   COPFB.CI_DATA0

CAL  COPFB

LD   COPFB.CS_CONFIRM
ST   CS_CONFIRM                    ** Conferma comando eseguito

LD   COPFB.CO_ERROR
ST   CO_ERROR                      ** Codice di errore

LD   COPFB.CO_ERRORINFO
ST   CO_ERRORINFO                  ** Informazioni aggiuntive su errore

END_FUNCTION_BLOCK

(* ---- CAP_EMP.plc ---- *)
*******************************************************************************
*   CAP_PREC.PLC
*   ESAutomotion
*   LASER machine
*******************************************************************************
VAR
#include "Cnc.inc"
#include "RemContr.inc"
***BTN_START_CALIB       AT %cButton0.0;     * Calibration START button
CapacitiveSimulated      AT %cOpt0.0;        * Capacitive simulated
IncStepQuota:            DWORD;  * Quota di incremento per controllo calibrazione
END_VAR

VAR_IN_OUT

#include "mem.inc"

BTN_START_CALIB         AT %cButton0.0;     * Calibration START button

CURVE_Y_P0              AT %rPlc10;
CURVE_Y_P1              AT %rPlc11;
CURVE_Y_P2              AT %rPlc12;
CURVE_Y_P3              AT %rPlc13;
CURVE_Y_P4              AT %rPlc14;
CURVE_Y_P5              AT %rPlc15;
CURVE_Y_P6              AT %rPlc16;
CURVE_Y_P7              AT %rPlc17;
CURVE_Y_P8              AT %rPlc18;
CURVE_Y_P9              AT %rPlc19;
CURVE_Y_P10             AT %rPlc20;

CURVE_X_P0              AT %rPlc21;
CURVE_X_P1              AT %rPlc22;
CURVE_X_P2              AT %rPlc23;
CURVE_X_P3              AT %rPlc24;
CURVE_X_P4              AT %rPlc25;
CURVE_X_P5              AT %rPlc26;
CURVE_X_P6              AT %rPlc27;
CURVE_X_P7              AT %rPlc28;
CURVE_X_P8              AT %rPlc29;
CURVE_X_P9              AT %rPlc30;
CURVE_X_P10             AT %rPlc31;

END_VAR

#include "Iol.inc"
#include "Cap_Prec.inc"

*******************************************************************************
*   CAPACITIVE: PROCON
*       %Capacitive[] structure used
*******************************************************************************
FUNCTION_BLOCK CAP_EMP
VAR_INPUT
xEmission:      BOOL;           * Emission command
xEmp_sensor:    DWORD;          * capacitive value
END_VAR

VAR_OUTPUT
yErr:           DWORD;          * error
yMsg:           DWORD;          * msg
yExeCalib:      BOOL;           * Calibration requested
yTipTouch:      BOOL;           * Tip touch signal without filter
yFar:           BOOL;
END_VAR

VAR
TipTouchNoFilered:      BOOL;   * Tip touch signal not filtered
CalibRequest:           BOOL;   * Calib request
CALIBRAZIONE_RUN:       BOOL;   * Programma calibrazione in corso
CALIBRAZIONE_ON:        BOOL;   * Ciclo calibrazione attivo
TIP_TOUCH:              BOOL;   * Tip touch intervenuto
BODY_TOUCH:             BOOL;   * Body touch intervenuto
NOZZLE_LOST:            BOOL;   * Ugello perso intervenuto
Strobe_Funz_M492:       BOOL;   * Nozzle verify
Tip_Touch_Status:       BOOL;
FilterTipTouch:         DWORD;  * Tip touch dynamic filter
TON_CALIBR:             TON;    * Ritardo verifica durata max calibrazione
TON_TIPTOUCH:           TON;    * Filtro Tip Touch laser mech
TON_ECAT:               TON;    * Ecatrun
R_TRIG492:              R_TRIG;
F_TRIG_LAS_OFF:         F_TRIG;
TP_DIS_TIP_TIPTOUCH:    TP;
RTRIG_REQUEST:          R_TRIG;
FT_PRGRUN:              F_TRIG;
* Remote Controller
RTRIG_CALIB:            R_TRIG;
END_VAR
*******************************************************************************

***************************************
*   Calibration request
***************************************
CAL  FT_PRGRUN(CLK=PRGRUN_CN0)     ** M0.0 cn0.rc8.0  Programma in corso
CAL  RTRIG_REQUEST(CLK=BTN_START_CALIB) ** Calibration START button
CAL  RTRIG_CALIB(CLK:=RemContrCalib) ** Xhc_Puls.12 Execute calibration

LD   RTRIG_REQUEST.Q
OR   RTRIG_CALIB.Q                 ** Xhc_Puls.12 Execute calibration)
AND  MACC_TARATA                   ** (gPlc0.9)Assi tarati
OR   CalibRequest                  ** Calib request
S    CalibRequest                  ** Calib request

LD   M30_CN0                       ** M0.13 M30:EndProgram CN0
OR   MACC_ALARM                    ** (gPlc0.10)Macchina in allarme
OR   RESET_ALLARMI                 ** M100.4  Cancellazione allarmi attiva
OR   FT_PRGRUN.Q
R    CalibRequest                  ** Calib request

LD   CalibRequest                  ** Calib request
ST   CALIBRAZIONE_RUN              ** Programma calibrazione in corso
ST   yMsg.0
ST   yExeCalib                     ** Calibration requested

***************************************
*   Calibrazione running
***************************************
LD   CalibRequest
ANDN RESET_MACCHINA                ** M100.2  Reset macchina
ST   CALIBRAZIONE_ON               ** Ciclo calibrazione attivo

LDN  MACCHINA_OK                   ** M100.1  Macchina OK
OR   RESET_MACCHINA                ** M100.2  Reset macchina
R    O_CALIBRA_REQ_A3              ** Calibration request
R    O_STROBE_A7                   ** Strobe

***************************************
*   TIP TOUCH
***************************************
LD   xEmp_sensor
LE   %EmConfig.mincapval
ST   Tip_Touch_Status

LD   %TsCalib1.targ_b_axis
SUB  1000
LT   %ax33.ra4
AND  CalibRequest
JMPCN TIPTOUCH15BVL
     LD   xEmp_sensor
     LE   %EmConfig.capval1
     ST   Tip_Touch_Status
TIPTOUCH15BVL:

LD   %TsCalib2.targ_b_axis
SUB  1000
LT   %ax33.ra4
AND  CalibRequest
JMPCN TIPTOUCH30BVL
     LD   xEmp_sensor
     LE   %EmConfig.capval2
     ST   Tip_Touch_Status
TIPTOUCH30BVL:

LD   %TsCalib3.targ_b_axis
SUB  1000
LT   %ax33.ra4
AND  CalibRequest
JMPCN TIPTOUCH45BVL
     LD   xEmp_sensor
     LE   %EmConfig.capval3
     ST   Tip_Touch_Status
TIPTOUCH45BVL:

LD   Tip_Touch_Status
OR (
LD   %M68.0 * TODO !!!!
AND (
LD   PLC_SIMULATED
EQ   1
)
)
ST   TipTouchNoFilered             ** Tip touch signal not filtered
ST   yTipTouch

LD   xEmp_sensor
GT   %EmConfig.FARcapval_Ang
ST   yFar

LD   TipTouchFilter                ** (rLsGui41) tip touch filter (msec)
ST   FilterTipTouch                ** Tip touch dynamic filter

LDN  PRGRUN_CN0                    ** M0.0 cn0.rc8.0  Programma in corso
OR   ReqCapacitveTest              ** (gPlc13.27) Capacitive test request
JMPCN no_calc_tip_touch_filt
LD   0
ST   FilterTipTouch                ** Tip touch dynamic filter
no_calc_tip_touch_filt:

CAL  F_TRIG_LAS_OFF(CLK:=xEmission) ** Emission command
CAL  TP_DIS_TIP_TIPTOUCH(IN:=F_TRIG_LAS_OFF.Q, PT:=300)
CAL  TON_TIPTOUCH(IN=TipTouchNoFilered,PT=FilterTipTouch) ** Filtro Tip Touch laser mech
CAL  TON_ECAT(IN=%ecat_ring.ec_status.31,PT=3000) **Ecatrun
LD   TON_TIPTOUCH.Q
ANDN InibTipTouchAllarm            ** M100.22 Inibizione allarme Tip Touch per restart ciclo
ANDN TipTouchDisable               ** (LsPlc71.0) TipTouchDisable (ritardato)
ANDN CALIBRAZIONE_RUN
ANDN TP_DIS_TIP_TIPTOUCH.Q
ANDN DisabTipTouch                  * singfc (G3300 / G3301)
AND (
LDN  CALIBRATION_CHECK              * (C26.0) Calibration control in run
OR (
LD   CALIBRATION_CHECK              * (C26.0) Calibration control in run
ANDN ISOTipTouchDisable             * (C26.3) Disabilita tip touch da ISO
)
)
AND  TON_ECAT.Q
ST   TIP_TOUCH                     ** Tip touch intervenuto
S    yErr.0

LD   RESET_ALLARMI                 ** M100.4  Cancellazione allarmi attiva
OR(
     LD  ButtClearAlarm                 ** (gGui23.0) Clear alarm interface push-button
     OR  RemContrCancAlarm			   * Xhc_Puls.31 Clear alarm
     AND (
     LD  PRGSTOP_CN0                    ** (cn0.rc8.1)  Programma interrotto CN0
     ORN PRGRUN_CN0                     ** M0.0 cn0.rc8.0  Programma in corso
     )
)
OR(
LD   Pul_Start                     ** (gPlc0.1)Start pushbutton
ANDN TIP_TOUCH                     ** Tip touch intervenuto
)
OR   InibTipTouchAllarm            ** M100.22 Inibizione allarme Tip Touch per restart ciclo
R    yErr.0

***************************************
*   Allarme: Tempo massimo calibrazione sensore capacitivo
***************************************
CAL  TON_CALIBR(IN=CALIBRAZIONE_ON,PT=200000) ** Ritardo verifica durata max calibrazione
LD   TON_CALIBR.Q        ** Trascorso tempo massimo per Calibrazione sensore capacitivo
S    yErr.3

LD   RESET_ALLARMI                 ** M100.4  Cancellazione allarmi attiva
R    yErr.3

***************************************
*   Allarme: Cavo interrotto da capacitivo
***************************************
*LD   xEmp_sensor                  ***cable cut
*EQ   0
*AND  TON_ECAT.Q
*S    yErr.4
*
*LD   RESET_ALLARMI                 ** M100.4  Cancellazione allarmi attiva
*R    yErr.4

*****************************************************************************
* Calibration Control
*****************************************************************************

LD   %SoftBtn0.20
JMPCN NoInitCurveCap

LD   0
ST   CURVE_Y_P0

*LD   409500                           * Capacitive sensor resolution 1mm
LD   AnalCapFeedback       *Capacitive analog resolution
MUL  1000
DIV  10000
ST   CURVE_Y_P1

*LD   409500                           * Capacitive sensor resolution 1mm
LD   AnalCapFeedback       *Capacitive analog resolution
MUL  1000
MUL  2
DIV  10000
ST   CURVE_Y_P2

*LD   409500                           * Capacitive sensor resolution 1mm
LD   AnalCapFeedback       *Capacitive analog resolution
MUL  1000
MUL  3
DIV  10000
ST   CURVE_Y_P3

*LD   409500                           * Capacitive sensor resolution 1mm
LD   AnalCapFeedback       *Capacitive analog resolution
MUL  1000
MUL  4
DIV  10000
ST   CURVE_Y_P4

*LD   409500                           * Capacitive sensor resolution 1mm
LD   AnalCapFeedback       *Capacitive analog resolution
MUL  1000
MUL  5
DIV  10000
ST   CURVE_Y_P5

*LD   409500                           * Capacitive sensor resolution 1mm
LD   AnalCapFeedback       *Capacitive analog resolution
MUL  1000
MUL  6
DIV  10000
ST   CURVE_Y_P6

*LD   409500                           * Capacitive sensor resolution 1mm
LD   AnalCapFeedback       *Capacitive analog resolution
MUL  1000
MUL  7
DIV  10000
ST   CURVE_Y_P7

*LD   409500                           * Capacitive sensor resolution 1mm
LD   AnalCapFeedback       *Capacitive analog resolution
MUL  1000
MUL  8
DIV  10000
ST   CURVE_Y_P8

*LD   409500                           * Capacitive sensor resolution 1mm
LD   AnalCapFeedback       *Capacitive analog resolution
MUL  1000
MUL  9
DIV  10000
ST   CURVE_Y_P9

*LD   409500                           * Capacitive sensor resolution 1mm
LD   AnalCapFeedback       *Capacitive analog resolution
MUL  1000
MUL  10
DIV  10000
ST   CURVE_Y_P10

NoInitCurveCap:

LD   1000
ST   IncStepQuota

LD   %LSRCostK31
EQ   20000
JMPCN SetTenMM

LD   2000
ST   IncStepQuota

SetTenMM:

LD   0
ST   CURVE_X_P0

LD   CURVE_X_P0
ADD  IncStepQuota
ST   CURVE_X_P1

LD   CURVE_X_P1
ADD  IncStepQuota
ST   CURVE_X_P2

LD   CURVE_X_P2
ADD  IncStepQuota
ST   CURVE_X_P3

LD   CURVE_X_P3
ADD  IncStepQuota
ST   CURVE_X_P4

LD   CURVE_X_P4
ADD  IncStepQuota
ST   CURVE_X_P5

LD   CURVE_X_P5
ADD  IncStepQuota
ST   CURVE_X_P6

LD   CURVE_X_P6
ADD  IncStepQuota
ST   CURVE_X_P7

LD   CURVE_X_P7
ADD  IncStepQuota
ST   CURVE_X_P8

LD   CURVE_X_P8
ADD  IncStepQuota
ST   CURVE_X_P9

LD   CURVE_X_P9
ADD  IncStepQuota
ST   CURVE_X_P10

* Questo per evitare di modificare la curva trovata

LD   0
ST   %rPlc32
LD   %LsIso90
ST   %rPlc33
LD   %LsIso91
ST   %rPlc34
LD   %LsIso92
ST   %rPlc35
LD   %LsIso93
ST   %rPlc36
LD   %LsIso94
ST   %rPlc37
LD   %LsIso95
ST   %rPlc38
LD   %LsIso96
ST   %rPlc39
LD   %LsIso97
ST   %rPlc40
LD   %LsIso98
ST   %rPlc41
LD   %LsIso99
ST   %rPlc42

*******************************************************************************
*   HMI
*******************************************************************************

LD   yTipTouch
ST   %cLeds0.1

LD   yErr.4                        ***Cable cut
ST   %cLeds0.2

END_FUNCTION_BLOCK

(* ---- CAP_Prec.plc ---- *)
*******************************************************************************
*   CAP_PREC.PLC
*   ESAutomotion
*   LASER machine
*******************************************************************************
VAR
#include "Cnc.inc"
#include "RemContr.inc"
***BTN_START_CALIB         AT %cButton0.0;     * Calibration START button
CapacitiveSimulated     AT %cOpt0.0;        * Capacitive simulated
IncStepQuota:            DWORD;  * Quota di incremento per controllo calibrazione
END_VAR

VAR_IN_OUT

#include "mem.inc"

BTN_START_CALIB         AT %cButton0.0;     * Calibration START button

CURVE_Y_P0              AT %rPlc10;
CURVE_Y_P1              AT %rPlc11;
CURVE_Y_P2              AT %rPlc12;
CURVE_Y_P3              AT %rPlc13;
CURVE_Y_P4              AT %rPlc14;
CURVE_Y_P5              AT %rPlc15;
CURVE_Y_P6              AT %rPlc16;
CURVE_Y_P7              AT %rPlc17;
CURVE_Y_P8              AT %rPlc18;
CURVE_Y_P9              AT %rPlc19;
CURVE_Y_P10             AT %rPlc20;

CURVE_X_P0              AT %rPlc21;
CURVE_X_P1              AT %rPlc22;
CURVE_X_P2              AT %rPlc23;
CURVE_X_P3              AT %rPlc24;
CURVE_X_P4              AT %rPlc25;
CURVE_X_P5              AT %rPlc26;
CURVE_X_P6              AT %rPlc27;
CURVE_X_P7              AT %rPlc28;
CURVE_X_P8              AT %rPlc29;
CURVE_X_P9              AT %rPlc30;
CURVE_X_P10             AT %rPlc31;

END_VAR

#include "Iol.inc"
#include "Cap_Prec.inc"

*******************************************************************************
*   CAPACITIVE: PROCON
*       %Capacitive[] structure used
*******************************************************************************
FUNCTION_BLOCK CAP_PREC
VAR_INPUT
xEmission:      BOOL;           * Emission command
END_VAR

VAR_OUTPUT
yErr:           DWORD;          * error
yMsg:           DWORD;          * msg
yExeCalib:      BOOL;           * Calibration requested
yTipTouch:      BOOL;           * Tip touch signal without filter
END_VAR

VAR
TipTouchNoFilered:      BOOL;   * Tip touch signal not filtered
CalibRequest:           BOOL;   * Calib request
CALIBRAZIONE_RUN:       BOOL;   * Programma calibrazione in corso
CALIBRAZIONE_ON:        BOOL;   * Ciclo calibrazione attivo
TIP_TOUCH:              BOOL;   * Tip touch intervenuto
BODY_TOUCH:             BOOL;   * Body touch intervenuto
NOZZLE_LOST:            BOOL;   * Ugello perso intervenuto
Strobe_Funz_M492:       BOOL;   * Nozzle verify
FilterTipTouch:         DWORD;  * Tip touch dynamic filter
TON_CALIBR:             TON;    * Ritardo verifica durata max calibrazione
TON_TIPTOUCH:           TON;    * Filtro Tip Touch laser mech
R_TRIG492:              R_TRIG;
F_TRIG_LAS_OFF:         F_TRIG;
TP_DIS_TIP_TIPTOUCH:    TP;
RTRIG_REQUEST:          R_TRIG;
FT_PRGRUN:              F_TRIG;
* Remote Controller
RTRIG_CALIB:            R_TRIG;
END_VAR
*******************************************************************************

***************************************
*   Calibration request
***************************************
CAL  FT_PRGRUN(CLK=PRGRUN_CN0)     ** M0.0 cn0.rc8.0  Programma in corso
CAL  RTRIG_REQUEST(CLK=BTN_START_CALIB) ** Calibration START button
CAL  RTRIG_CALIB(CLK:=RemContrCalib) ** Xhc_Puls.12 Execute calibration

LD   RTRIG_REQUEST.Q
OR   RTRIG_CALIB.Q                 ** Xhc_Puls.12 Execute calibration)
AND  MACC_TARATA                   ** (gPlc0.9)Assi tarati
OR   CalibRequest                  ** Calib request
S    CalibRequest                  ** Calib request

LD   M30_CN0                       ** M0.13 M30:EndProgram CN0
OR   MACC_ALARM                    ** (gPlc0.10)Macchina in allarme
OR   RESET_ALLARMI                 ** M100.4  Cancellazione allarmi attiva
OR   FT_PRGRUN.Q
R    CalibRequest                  ** Calib request

LD   CalibRequest                  ** Calib request
ST   CALIBRAZIONE_RUN              ** Programma calibrazione in corso
ST   yMsg.0
ST   yExeCalib                     ** Calibration requested

***************************************
*   Calibrazione running
***************************************
LD   O_CALIBRA_REQ_A3              ** Calibration request
ANDN I_READY_A13                   ** Ready
ANDN RESET_MACCHINA                ** M100.2  Reset macchina
ST   CALIBRAZIONE_ON               ** Ciclo calibrazione attivo

LDN  MACCHINA_OK                   ** M100.1  Macchina OK
OR   RESET_MACCHINA                ** M100.2  Reset macchina
R    O_CALIBRA_REQ_A3              ** Calibration request
R    O_STROBE_A7                   ** Strobe

***************************************
*   TIP TOUCH
***************************************
LD   I_TIP_BODY_TOUCH_A11          ** Tip\Body Touch or Nozzle_Lost (TIP TOUCH:A11=1,A14=0,A15=0)
ANDN I_BODY_TOUCH_A14              ** Body touch (A11=1,A14=1,A15=0)
ANDN I_NOZZLE_LOST_A15             ** Nozzle Lost/Pos reached (NOZZLE LOST:A11=1,A14=0,A15=1)
OR (
LD   %M68.0 * TODO !!!!
AND (
LD   PLC_SIMULATED
EQ   1
)
)
ST   TipTouchNoFilered             ** Tip touch signal not filtered
ST   yTipTouch

LD   TipTouchFilter                ** (rLsGui41) tip touch filter (msec)
ST   FilterTipTouch                ** Tip touch dynamic filter

LDN  PRGRUN_CN0                    ** M0.0 cn0.rc8.0  Programma in corso
OR   ReqCapacitveTest              ** (gPlc13.27) Capacitive test request
JMPCN no_calc_tip_touch_filt
LD   0
ST   FilterTipTouch                ** Tip touch dynamic filter
no_calc_tip_touch_filt:

CAL  F_TRIG_LAS_OFF(CLK:=xEmission) ** Emission command
CAL  TP_DIS_TIP_TIPTOUCH(IN:=F_TRIG_LAS_OFF.Q, PT:=300)
CAL  TON_TIPTOUCH(IN=TipTouchNoFilered,PT=FilterTipTouch) ** Filtro Tip Touch laser mech

LD   TON_TIPTOUCH.Q
ANDN InibTipTouchAllarm            ** M100.22 Inibizione allarme Tip Touch per restart ciclo
ANDN TipTouchDisable               ** (LsPlc71.0) TipTouchDisable (ritardato)
ANDN O_CALIBRA_REQ_A3              ** Calibration request
ANDN TP_DIS_TIP_TIPTOUCH.Q
ANDN DisabTipTouch                  * singfc (G3300 / G3301)
AND (
LDN  CALIBRATION_CHECK              * (C26.0) Calibration control in run
OR (
LD   CALIBRATION_CHECK              * (C26.0) Calibration control in run
ANDN ISOTipTouchDisable             * (C26.3) Disabilita tip touch da ISO
)
)
ST   TIP_TOUCH                     ** Tip touch intervenuto
S    yErr.0

LD   RESET_ALLARMI                 ** M100.4  Cancellazione allarmi attiva
OR(
LD   Pul_Start                     ** (gPlc0.1)Start pushbutton
ANDN TIP_TOUCH                     ** Tip touch intervenuto
)
OR   InibTipTouchAllarm            ** M100.22 Inibizione allarme Tip Touch per restart ciclo
R    yErr.0

***************************************
*   BODY TOUCH
***************************************
LD   I_TIP_BODY_TOUCH_A11          ** Tip\Body Touch or Nozzle_Lost (TIP TOUCH:A11=1,A14=0,A15=0)
AND  I_BODY_TOUCH_A14              ** Body touch (A11=1,A14=1,A15=0)
ANDN I_NOZZLE_LOST_A15             ** Nozzle Lost/Pos reached (NOZZLE LOST:A11=1,A14=0,A15=1)
ST   BODY_TOUCH                    ** Body touch intervenuto

LD   BODY_TOUCH                    ** Body touch intervenuto
S    yErr.1

LD   RESET_ALLARMI                 ** M100.4  Cancellazione allarmi attiva
R    yErr.1

***************************************
*   NOZZLE LOST
***************************************
LD   I_TIP_BODY_TOUCH_A11          ** Tip\Body Touch or Nozzle_Lost (TIP TOUCH:A11=1,A14=0,A15=0)
ANDN I_BODY_TOUCH_A14              ** Body touch (A11=1,A14=1,A15=0)
AND  I_NOZZLE_LOST_A15             ** Nozzle Lost/Pos reached (NOZZLE LOST:A11=1,A14=0,A15=1)
ST   NOZZLE_LOST                   ** Ugello perso intervenuto

***************************************
*   M492 Verifica presenza NOZZLE LOST
***************************************
LD   %cn0.rc9                        ** Channel 0 M-Functions register
EQ   492
AND  %cn0.rc8.4                    ** Channel 0 M-Functions Strobe
OR   VerNozzlelost                 ** (TstP15.0) Verifica NOZZLE LOST
ST   Strobe_Funz_M492              ** Nozzle verify

CAL  R_TRIG492(CLK=Strobe_Funz_M492) ** Nozzle verify

LD   R_TRIG492.Q                    **Strobe funzione M492
AND  NOZZLE_LOST                   ** Ugello perso intervenuto
OR   NOZZLE_LOST
ANDN CALIBRAZIONE_RUN              ** Programma calibrazione in corso
S    yErr.2

LD   RESET_ALLARMI                 ** M100.4  Cancellazione allarmi attiva
OR(
LD   Pul_Start                     ** (gPlc0.1)Start pushbutton
ANDN NOZZLE_LOST                   ** Ugello perso intervenuto
)
R    yErr.2

***************************************
*   Allarme: Tempo massimo calibrazione sensore capacitivo
***************************************
CAL  TON_CALIBR(IN=CALIBRAZIONE_ON,PT=120000) ** Ritardo verifica durata max calibrazione
LD   TON_CALIBR.Q        ** Trascorso tempo massimo per Calibrazione sensore capacitivo
S    yErr.3

LD   RESET_ALLARMI                 ** M100.4  Cancellazione allarmi attiva
R    yErr.3

***************************************
*   Allarme: Cavo interrotto da capacitivo
***************************************
LD   I_CABLE_CUT_A12               ** Cable cut
S    yErr.4

LD   RESET_ALLARMI                 ** M100.4  Cancellazione allarmi attiva
R    yErr.4

*******************************************************************************
*   Message: check if there is a wrong condition with FAR input and capacitive
*   If FAR=1 and capacitive not 10V means there are some problem with the capacitive
*******************************************************************************
LD   %LSRPlcOp0.20                 ** FAR INPUT management enabled
AND  I_FAR_A10                     ** Far away
AND (
LD   IA_A18_19_DIST_LINEAR         ** Capacitive sensor
LT   (
LD   AnalCapFeedback       *Capacitive analog resolution
DIV  2
)
)
ST   yErr.5                  ** Check FAR e/o CAPACITIVE

LD   CapacitiveSimulated           ** Capacitive simulated
JMPCN NoSimC

LD   0
ST   yErr                          ** error
ST   yMsg                          ** msg

LD   ALWAYS_ONE                    ** PLCFLAGS.1  Flag sempre stato on
ST   yMsg.1                     * msg capacitive simulated

NoSimC:

*****************************************************************************
* Calibration Control
*****************************************************************************

LD   %SoftBtn0.20
JMPCN NoInitCurveCap

LD   0
ST   CURVE_Y_P0

*LD   409500                           * Capacitive sensor resolution 1mm
LD   AnalCapFeedback       *Capacitive analog resolution
MUL  1000
DIV  10000
ST   CURVE_Y_P1

*LD   409500                           * Capacitive sensor resolution 1mm
LD   AnalCapFeedback       *Capacitive analog resolution
MUL  1000
MUL  2
DIV  10000
ST   CURVE_Y_P2

*LD   409500                           * Capacitive sensor resolution 1mm
LD   AnalCapFeedback       *Capacitive analog resolution
MUL  1000
MUL  3
DIV  10000
ST   CURVE_Y_P3

*LD   409500                           * Capacitive sensor resolution 1mm
LD   AnalCapFeedback       *Capacitive analog resolution
MUL  1000
MUL  4
DIV  10000
ST   CURVE_Y_P4

*LD   409500                           * Capacitive sensor resolution 1mm
LD   AnalCapFeedback       *Capacitive analog resolution
MUL  1000
MUL  5
DIV  10000
ST   CURVE_Y_P5

*LD   409500                           * Capacitive sensor resolution 1mm
LD   AnalCapFeedback       *Capacitive analog resolution
MUL  1000
MUL  6
DIV  10000
ST   CURVE_Y_P6

*LD   409500                           * Capacitive sensor resolution 1mm
LD   AnalCapFeedback       *Capacitive analog resolution
MUL  1000
MUL  7
DIV  10000
ST   CURVE_Y_P7

*LD   409500                           * Capacitive sensor resolution 1mm
LD   AnalCapFeedback       *Capacitive analog resolution
MUL  1000
MUL  8
DIV  10000
ST   CURVE_Y_P8

*LD   409500                           * Capacitive sensor resolution 1mm
LD   AnalCapFeedback       *Capacitive analog resolution
MUL  1000
MUL  9
DIV  10000
ST   CURVE_Y_P9

*LD   409500                           * Capacitive sensor resolution 1mm
LD   AnalCapFeedback       *Capacitive analog resolution
MUL  1000
MUL  10
DIV  10000
ST   CURVE_Y_P10

NoInitCurveCap:

LD   1000
ST   IncStepQuota

LD   %LSRCostK31
EQ   20000
JMPCN SetTenMM

LD   2000
ST   IncStepQuota

SetTenMM:

LD   0
ST   CURVE_X_P0

LD   CURVE_X_P0
ADD  IncStepQuota
ST   CURVE_X_P1

LD   CURVE_X_P1
ADD  IncStepQuota
ST   CURVE_X_P2

LD   CURVE_X_P2
ADD  IncStepQuota
ST   CURVE_X_P3

LD   CURVE_X_P3
ADD  IncStepQuota
ST   CURVE_X_P4

LD   CURVE_X_P4
ADD  IncStepQuota
ST   CURVE_X_P5

LD   CURVE_X_P5
ADD  IncStepQuota
ST   CURVE_X_P6

LD   CURVE_X_P6
ADD  IncStepQuota
ST   CURVE_X_P7

LD   CURVE_X_P7
ADD  IncStepQuota
ST   CURVE_X_P8

LD   CURVE_X_P8
ADD  IncStepQuota
ST   CURVE_X_P9

LD   CURVE_X_P9
ADD  IncStepQuota
ST   CURVE_X_P10

* Questo per evitare di modificare la curva trovata

LD   0
ST   %rPlc32
LD   %LsIso90
ST   %rPlc33
LD   %LsIso91
ST   %rPlc34
LD   %LsIso92
ST   %rPlc35
LD   %LsIso93
ST   %rPlc36
LD   %LsIso94
ST   %rPlc37
LD   %LsIso95
ST   %rPlc38
LD   %LsIso96
ST   %rPlc39
LD   %LsIso97
ST   %rPlc40
LD   %LsIso98
ST   %rPlc41
LD   %LsIso99
ST   %rPlc42

*******************************************************************************
*   HMI
*******************************************************************************
LD   I_FAR_A10                     ** Far away
ST   %cLeds0.0
LD   I_TIP_BODY_TOUCH_A11          ** Tip\Body Touch or Nozzle_Lost (TIP TOUCH:A11=1,A14=0,A15=0)
ST   %cLeds0.1
LD   I_CABLE_CUT_A12               ** Cable cut
ST   %cLeds0.2
LD   I_READY_A13                   ** Ready
ST   %cLeds0.3
LD   I_BODY_TOUCH_A14              ** Body touch (A11=1,A14=1,A15=0)
ST   %cLeds0.4
LD   I_NOZZLE_LOST_A15             ** Nozzle Lost/Pos reached (NOZZLE LOST:A11=1,A14=0,A15=1)
ST   %cLeds0.5

LD   O_CALIBRA_REQ_A3              ** Calibration request
ST   %cLeds1.0
LD   O_STROBE_A7                   ** Strobe
ST   %cLeds1.1
LD   O_SELCHAR_BIT0_A4             ** Selecting the calibrated characteristic curve (1-8)
ST   %cLeds1.2
LD   O_SELCHAR_BIT1_A5             ** Selecting the calibrated characteristic curve (1-8)
ST   %cLeds1.3
LD   O_SELCHAR_BIT2_A6             ** Selecting the calibrated characteristic curve (1-8)
ST   %cLeds1.4

END_FUNCTION_BLOCK
